(* Schneider Machine Expert - Basic project 4pompe_alternanza_1allavolta_2soglie, file version 3.0.0.0 *)
(* ProjectInformations: Name=New project *)

HARDWARE
  Cpu 0: TM221C40R
  EthernetConfiguration: NetworkName=M221, IpAllocationMode=FixedAddress, IpAddress=0.0.0.0, SubnetMask=0.0.0.0
  SerialLineConfiguration: Baud=Baud19200, Parity=ParityEven, DataBits=DataBits8, StopBits=StopBits1, PhysicalMedium=PhysicalMediumRs485, TransmissionMode=TransmissionModeModbusRtu, SlaveId=1, Addressing=SlaveAddressing
  MastTask: UsePeriodScanMode=false, PeriodScan=100
  FastTask: Period=255
  CpuBehavior: StartingMode=StartAsPreviousState, AutoSaveRamOnEeprom=true, WatchdogPeriod=250

SYMBOLS  (address, symbol, comment, settings)
  %M0       P1_USABILE
  %M1       P2_USABILE
  %M2       P3_USABILE
  %M3       P4_USABILE
  %MW0      ULTIMA_POMPA_CMD
  %MW1      PROSSIMA_POMPA_CANDIDATA
  %I0.0     P1_AUTO
  %I0.1     P1_MOTO
  %I0.2     P1_ANOMALIA
  %I0.3     P2_AUTO
  %I0.4     P2_MOTO
  %I0.5     P2_ANOMALIA
  %I0.6     P3_AUTO
  %I0.7     P3_MOTO
  %I0.8     P3_ANOMALIA
  %I0.9     P4_AUTO
  %I0.10    P4_MOTO
  %I0.11    P4_ANOMALIA
  %I0.12    LVL_MIN
  %I0.13    LVL_MAX
  %Q0.0     P1_CMD
  %Q0.1     P2_CMD
  %Q0.2     P3_CMD
  %Q0.3     P4_CMD

POU New POU
  (* SectionNumber=1 *)

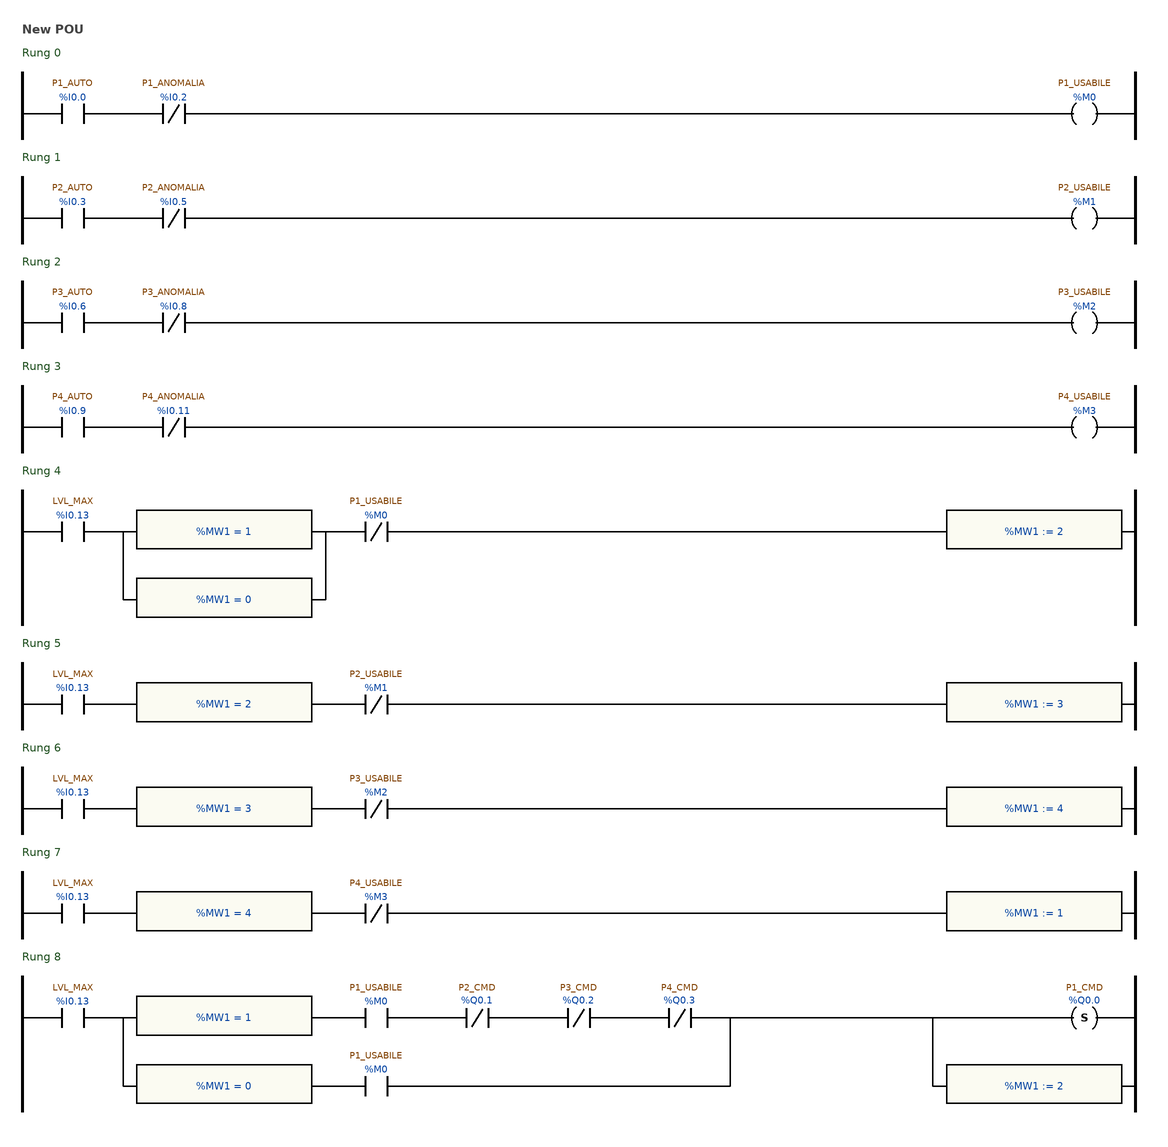

// Rung 0
  LD %I0.0                (* P1_AUTO *)
  ANDN %I0.2              (* P1_ANOMALIA *)
  ST %M0                  (* P1_USABILE *)
  // as ST:
  //   P1_USABILE := P1_AUTO AND NOT P1_ANOMALIA;

// Rung 1
  LD %I0.3                (* P2_AUTO *)
  ANDN %I0.5              (* P2_ANOMALIA *)
  ST %M1                  (* P2_USABILE *)
  // as ST:
  //   P2_USABILE := P2_AUTO AND NOT P2_ANOMALIA;

// Rung 2
  LD %I0.6                (* P3_AUTO *)
  ANDN %I0.8              (* P3_ANOMALIA *)
  ST %M2                  (* P3_USABILE *)
  // as ST:
  //   P3_USABILE := P3_AUTO AND NOT P3_ANOMALIA;

// Rung 3
  LD %I0.9                (* P4_AUTO *)
  ANDN %I0.11             (* P4_ANOMALIA *)
  ST %M3                  (* P4_USABILE *)
  // as ST:
  //   P4_USABILE := P4_AUTO AND NOT P4_ANOMALIA;

// Rung 4
  LD %I0.13               (* LVL_MAX *)
  AND( [ %MW1 = 1 ]       (* PROSSIMA_POMPA_CANDIDATA *)
  OR [ %MW1 = 0 ]         (* PROSSIMA_POMPA_CANDIDATA *)
  )
  ANDN %M0                (* P1_USABILE *)
  [ %MW1 := 2 ]           (* PROSSIMA_POMPA_CANDIDATA *)
  // as ST:
  //   IF LVL_MAX AND (PROSSIMA_POMPA_CANDIDATA = 1 OR PROSSIMA_POMPA_CANDIDATA = 0) AND NOT P1_USABILE THEN PROSSIMA_POMPA_CANDIDATA := 2; END_IF;

// Rung 5
  LD %I0.13               (* LVL_MAX *)
  AND [ %MW1 = 2 ]        (* PROSSIMA_POMPA_CANDIDATA *)
  ANDN %M1                (* P2_USABILE *)
  [ %MW1 := 3 ]           (* PROSSIMA_POMPA_CANDIDATA *)
  // as ST:
  //   IF LVL_MAX AND PROSSIMA_POMPA_CANDIDATA = 2 AND NOT P2_USABILE THEN PROSSIMA_POMPA_CANDIDATA := 3; END_IF;

// Rung 6
  LD %I0.13               (* LVL_MAX *)
  AND [ %MW1 = 3 ]        (* PROSSIMA_POMPA_CANDIDATA *)
  ANDN %M2                (* P3_USABILE *)
  [ %MW1 := 4 ]           (* PROSSIMA_POMPA_CANDIDATA *)
  // as ST:
  //   IF LVL_MAX AND PROSSIMA_POMPA_CANDIDATA = 3 AND NOT P3_USABILE THEN PROSSIMA_POMPA_CANDIDATA := 4; END_IF;

// Rung 7
  LD %I0.13               (* LVL_MAX *)
  AND [ %MW1 = 4 ]        (* PROSSIMA_POMPA_CANDIDATA *)
  ANDN %M3                (* P4_USABILE *)
  [ %MW1 := 1 ]           (* PROSSIMA_POMPA_CANDIDATA *)
  // as ST:
  //   IF LVL_MAX AND PROSSIMA_POMPA_CANDIDATA = 4 AND NOT P4_USABILE THEN PROSSIMA_POMPA_CANDIDATA := 1; END_IF;

// Rung 8
  LD %I0.13               (* LVL_MAX *)
  AND( [ %MW1 = 1 ]       (* PROSSIMA_POMPA_CANDIDATA *)
  AND %M0                 (* P1_USABILE *)
  ANDN %Q0.1              (* P2_CMD *)
  ANDN %Q0.2              (* P3_CMD *)
  ANDN %Q0.3              (* P4_CMD *)
  OR( [ %MW1 = 0 ]        (* PROSSIMA_POMPA_CANDIDATA *)
  AND %M0                 (* P1_USABILE *)
  )
  )
  S %Q0.0                 (* P1_CMD *)
  [ %MW1 := 2 ]           (* PROSSIMA_POMPA_CANDIDATA *)
  // as ST:
  //   IF LVL_MAX AND (PROSSIMA_POMPA_CANDIDATA = 1 AND P1_USABILE AND NOT P2_CMD AND NOT P3_CMD AND NOT P4_CMD OR PROSSIMA_POMPA_CANDIDATA = 0 AND P1_USABILE) THEN P1_CMD := TRUE; END_IF;
  //   IF LVL_MAX AND (PROSSIMA_POMPA_CANDIDATA = 1 AND P1_USABILE AND NOT P2_CMD AND NOT P3_CMD AND NOT P4_CMD OR PROSSIMA_POMPA_CANDIDATA = 0 AND P1_USABILE) THEN PROSSIMA_POMPA_CANDIDATA := 2; END_IF;

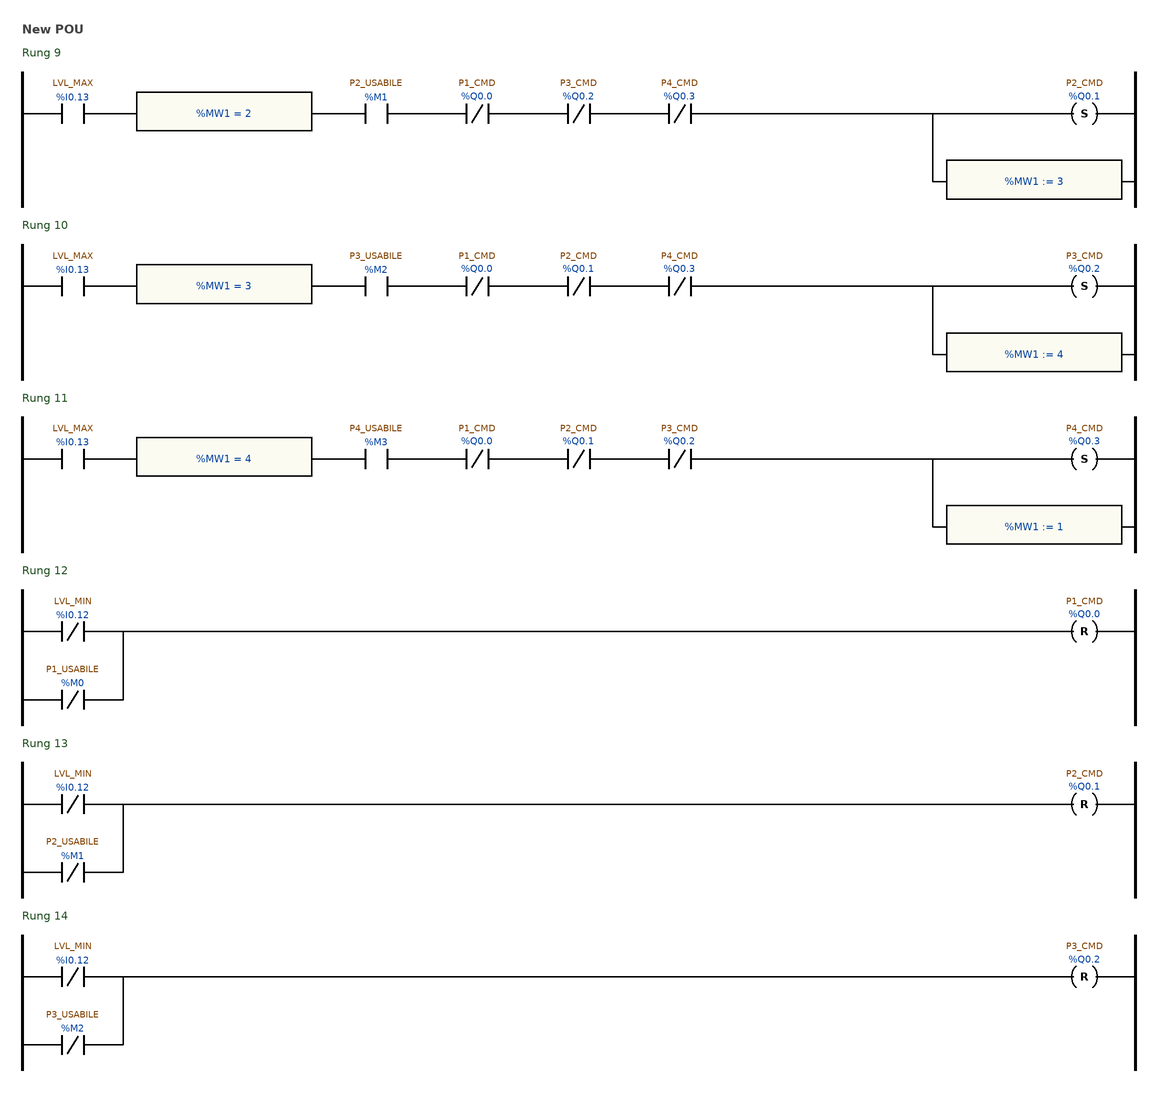

// Rung 9
  LD %I0.13               (* LVL_MAX *)
  AND [ %MW1 = 2 ]        (* PROSSIMA_POMPA_CANDIDATA *)
  AND %M1                 (* P2_USABILE *)
  ANDN %Q0.0              (* P1_CMD *)
  ANDN %Q0.2              (* P3_CMD *)
  ANDN %Q0.3              (* P4_CMD *)
  S %Q0.1                 (* P2_CMD *)
  [ %MW1 := 3 ]           (* PROSSIMA_POMPA_CANDIDATA *)
  // as ST:
  //   IF LVL_MAX AND PROSSIMA_POMPA_CANDIDATA = 2 AND P2_USABILE AND NOT P1_CMD AND NOT P3_CMD AND NOT P4_CMD THEN P2_CMD := TRUE; END_IF;
  //   IF LVL_MAX AND PROSSIMA_POMPA_CANDIDATA = 2 AND P2_USABILE AND NOT P1_CMD AND NOT P3_CMD AND NOT P4_CMD THEN PROSSIMA_POMPA_CANDIDATA := 3; END_IF;

// Rung 10
  LD %I0.13               (* LVL_MAX *)
  AND [ %MW1 = 3 ]        (* PROSSIMA_POMPA_CANDIDATA *)
  AND %M2                 (* P3_USABILE *)
  ANDN %Q0.0              (* P1_CMD *)
  ANDN %Q0.1              (* P2_CMD *)
  ANDN %Q0.3              (* P4_CMD *)
  S %Q0.2                 (* P3_CMD *)
  [ %MW1 := 4 ]           (* PROSSIMA_POMPA_CANDIDATA *)
  // as ST:
  //   IF LVL_MAX AND PROSSIMA_POMPA_CANDIDATA = 3 AND P3_USABILE AND NOT P1_CMD AND NOT P2_CMD AND NOT P4_CMD THEN P3_CMD := TRUE; END_IF;
  //   IF LVL_MAX AND PROSSIMA_POMPA_CANDIDATA = 3 AND P3_USABILE AND NOT P1_CMD AND NOT P2_CMD AND NOT P4_CMD THEN PROSSIMA_POMPA_CANDIDATA := 4; END_IF;

// Rung 11
  LD %I0.13               (* LVL_MAX *)
  AND [ %MW1 = 4 ]        (* PROSSIMA_POMPA_CANDIDATA *)
  AND %M3                 (* P4_USABILE *)
  ANDN %Q0.0              (* P1_CMD *)
  ANDN %Q0.1              (* P2_CMD *)
  ANDN %Q0.2              (* P3_CMD *)
  S %Q0.3                 (* P4_CMD *)
  [ %MW1 := 1 ]           (* PROSSIMA_POMPA_CANDIDATA *)
  // as ST:
  //   IF LVL_MAX AND PROSSIMA_POMPA_CANDIDATA = 4 AND P4_USABILE AND NOT P1_CMD AND NOT P2_CMD AND NOT P3_CMD THEN P4_CMD := TRUE; END_IF;
  //   IF LVL_MAX AND PROSSIMA_POMPA_CANDIDATA = 4 AND P4_USABILE AND NOT P1_CMD AND NOT P2_CMD AND NOT P3_CMD THEN PROSSIMA_POMPA_CANDIDATA := 1; END_IF;

// Rung 12
  LDN %I0.12              (* LVL_MIN *)
  ORN %M0                 (* P1_USABILE *)
  R %Q0.0                 (* P1_CMD *)
  // as ST:
  //   IF NOT LVL_MIN OR NOT P1_USABILE THEN P1_CMD := FALSE; END_IF;

// Rung 13
  LDN %I0.12              (* LVL_MIN *)
  ORN %M1                 (* P2_USABILE *)
  R %Q0.1                 (* P2_CMD *)
  // as ST:
  //   IF NOT LVL_MIN OR NOT P2_USABILE THEN P2_CMD := FALSE; END_IF;

// Rung 14
  LDN %I0.12              (* LVL_MIN *)
  ORN %M2                 (* P3_USABILE *)
  R %Q0.2                 (* P3_CMD *)
  // as ST:
  //   IF NOT LVL_MIN OR NOT P3_USABILE THEN P3_CMD := FALSE; END_IF;

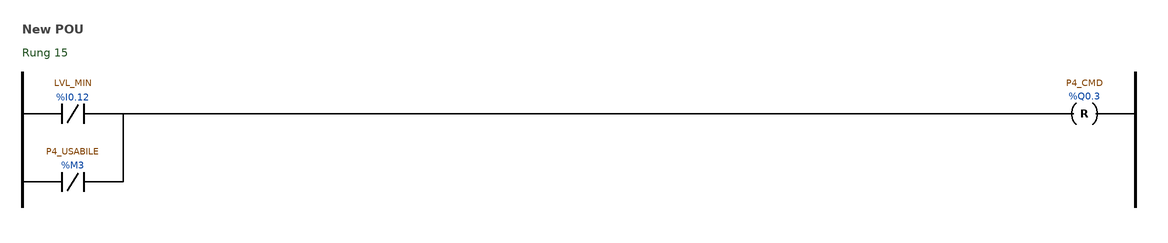

// Rung 15
  LDN %I0.12              (* LVL_MIN *)
  ORN %M3                 (* P4_USABILE *)
  R %Q0.3                 (* P4_CMD *)
  // as ST:
  //   IF NOT LVL_MIN OR NOT P4_USABILE THEN P4_CMD := FALSE; END_IF;
